FUNCTION_BLOCK TcpIp
VAR_INPUT
	
	bEnable : BOOL;
	stServerData : ST_ServerData;
	stClientData : ST_ClientData;
	
END_VAR
VAR_OUTPUT
END_VAR
VAR

	fbClientServerConnection : FB_ClientServerConnection;
	fbServerClientConnection : FB_ServerClientConnection;
	fbSocketSend : FB_SocketSend;
	fbSocketReceive : FB_SocketReceive;
	
	stepSendRoutine : UINT;
	stepReceiveRoutine : UINT;
	eMode : E_TcpIpMode;
	hSocket : T_HSOCKET;
	bResetConnection : BOOL;
END_VAR


fbSocketSend(
	sSrvNetId:= , 
	hSocket:= hSocket, 
	cbLen:= , 
	pSrc:= , 
	bExecute:= , 
	tTimeout:= , 
	bBusy=> , 
	bError=> , 
	nErrId=> );
	
fbSocketReceive(
	sSrvNetId:= , 
	hSocket:= hSocket, 
	cbLen:= , 
	pDest:= , 
	bExecute:= , 
	tTimeout:= , 
	bBusy=> , 
	bError=> , 
	nErrId=> , 
	nRecBytes=> );

CASE eMode OF

	TCP_IP_SERVER:
		F_CreateServerHnd(
			sSrvNetID := stServerData.sSrvNetID,
			bEnable := bEnable,
			sLocalHost := stServerData.sLocalHost,
			nLocalPort := stServerData.nLocalPort,
			nMode := stServerData.nMode,
			hServer := stServerData.hServer
		);
			
		fbServerClientConnection(
			hServer:= stServerData.hServer,
			eMode:= , 
			sRemoteHost:= , 
			nRemotePort:= , 
			bEnable:= bEnable, 
			tReconnect:= , 
			bBusy=> , 
			bError=> , 
			nErrID=> , 
			hSocket=> , 
			eState=> );
			
		IF 	fbServerClientConnection.eState = eSOCKET_DISCONNECTED 
			THEN
			
			fbServerClientConnection(
			hServer:= stServerData.hServer,
			eMode:= , 
			sRemoteHost:= , 
			nRemotePort:= , 
			bEnable:= FALSE, 
			tReconnect:= , 
			bBusy=> , 
			bError=> , 
			nErrID=> , 
			hSocket=> , 
			eState=> );
			
		END_IF
		
		hSocket := fbServerClientConnection.hSocket;	
		
	TCP_IP_CLIENT:
	
		fbClientServerConnection(
			sSrvNetID:= stClientData.sSrvNetID, 
			nMode:= stClientData.nMode, 
			sRemoteHost:= stClientData.sRemoteHost, 
			nRemotePort:= stClientData.nRemotePort, 
			bEnable:= bEnable, 
			tReconnect:= stClientData.tReconnect, 
			bBusy=> , 
			bError=> , 
			nErrId=> , 
			hSocket=> , 
			eState=> );
			
		IF 	bResetConnection
			THEN
			
			bResetConnection := FALSE;
			fbClientServerConnection(
				sSrvNetID:= stClientData.sSrvNetID, 
				nMode:= stClientData.nMode, 
				sRemoteHost:= stClientData.sRemoteHost, 
				nRemotePort:= stClientData.nRemotePort, 
				bEnable:= FALSE, 
				tReconnect:= stClientData.tReconnect, 
				bBusy=> , 
				bError=> , 
				nErrId=> , 
				hSocket=> , 
				eState=> );
		END_IF
		
		hSocket := fbClientServerConnection.hSocket;		
		
END_CASE

METHOD FB_init : BOOL
VAR_INPUT
	bInitRetains : BOOL; // if TRUE, the retain variables are initialized (warm start / cold start)
	bInCopyCode : BOOL;  // if TRUE, the instance afterwards gets moved into the copy code (online change)
	eMode : E_TcpIpMode;
END_VAR
THIS^.eMode := eMode;
END_METHOD

METHOD ReceiveSerializedObject : BOOL
VAR_INPUT
	cbLen      : UDINT;
   	pDest      : POINTER TO BYTE;
END_VAR
IF	fbClientServerConnection.eState = eSOCKET_CONNECTED
	OR fbServerClientConnection.eState = eSOCKET_CONNECTED
THEN
	CASE stepReceiveRoutine OF
	
		0: 
			fbSocketReceive.pDest := pDest;
			fbSocketReceive.cbLen := cbLen;
			fbSocketReceive.bExecute := TRUE;
			stepReceiveRoutine := 10;
			
		10:
		
			IF 	NOT fbSocketReceive.bBusy
				AND NOT fbSocketReceive.bError
				AND fbSocketReceive.nRecBytes = cbLen
				THEN
				
				fbSocketReceive.bExecute := FALSE;
				ReceiveSerializedObject := TRUE;
				stepReceiveRoutine := 0;
				
			ELSIF 	NOT fbSocketReceive.bBusy
					AND NOT fbSocketReceive.bError
					AND fbSocketReceive.nRecBytes = 0
					THEN
					
					fbSocketReceive.bExecute := FALSE;
					stepReceiveRoutine := 0;
					
			ELSIF	fbSocketReceive.bError
					THEN
		
					bResetConnection := TRUE;
					fbSocketReceive.bExecute := FALSE;
					stepReceiveRoutine := 0;			
			END_IF
			
	END_CASE
END_IF
END_METHOD

METHOD SendSerializedObject : BOOL
VAR_INPUT
	cbLen      : UDINT;
    pSrc       : POINTER TO BYTE;
END_VAR
IF 	fbClientServerConnection.eState = eSOCKET_CONNECTED
	OR fbServerClientConnection.eState = eSOCKET_CONNECTED
THEN
	CASE stepSendRoutine OF
	
		0: 
		
			fbSocketSend.pSrc := pSrc;
			fbSocketSend.cbLen := cbLen;
			fbSocketSend.bExecute := TRUE;
			stepSendRoutine := 10;
			
		10:
		
			IF 	NOT fbSocketSend.bBusy
				AND NOT fbSocketSend.bError
				
				THEN
				
				fbSocketSend.bExecute := FALSE;
				SendSerializedObject := TRUE;
				stepSendRoutine := 0;
				
			END_IF
			
	END_CASE
END_IF
END_METHOD

END_FUNCTION_BLOCK

(* stored: Version 1.1.0.1, ProductVersion 3.1.4024.2
   POU TcpIp: Id {326bedf4-567c-4c8e-8600-6115e82aa01f}, SpecialFunc None
   Method FB_init: Id {f48f49c3-fcc6-44bb-b969-21bcdbad80b9}
   Method ReceiveSerializedObject: Id {e008cc05-7d40-4df9-81df-2d00e6b0a968}
   Method SendSerializedObject: Id {8addfef6-b092-4f41-93ac-2b22dda4f562} *)
